// TwinCAT 3 PLC project Automation_BaseClasses
// Title: Automation base classes
// Company: PTW TUDa
// ProjectVersion: 0.1
// ProgramVersion: 3.1.4023.0
// project tree:
//   DUTs/0_Base Data Structs/ E_SystemControlState.TcDUT (not stored), E_SystemOperatingState.TcDUT (not stored), ST_Control.TcDUT (not stored), ST_ControlState.TcDUT (not stored), ST_ErrorState.TcDUT (not stored), ST_SetPointState.TcDUT, ST_SetSetPoint.TcDUT (not stored), ST_SystemState.TcDUT (not stored)
//   DUTs/Actor Data Structs/Pumps/ E_Liquids.TcTLEO, ST_PumpGrundfosMagna3SetParameters.TcDUT (not stored), ST_PumpGrundfosMagna3State.TcDUT (not stored)
//   DUTs/System Data Structs/ ST_SystemClimatizedRoomChillerSetParameters.TcDUT, ST_SystemClimatizedRoomChillerState.TcDUT
//   POUs/0_Base Clases/ FB_Actor2Point.TcPOU, FB_ActorContinous.TcPOU (not stored), FB_SystemContinous.TcPOU
//   POUs/Actors/ FB_PumpGrundfosMagna3.TcPOU
//   POUs/Sensors/ FB_AnalogSensor.TcPOU, FB_Flow_Sensor.TcPOU, FB_Pressure_Sensor.TcPOU, FB_Temp_Sensor.TcPOU (not stored)

// ---- DUTs/0_Base Data Structs/ST_SetPointState.TcDUT
{attribute 'OPC.UA.DA.StructuredType' := '1'}
TYPE ST_SetPointState :
STRUCT
	fOperatingPoint	: REAL; //current operating point
	fSetPoint		: REAL; //current set point
	aSetPointLimits	: ARRAY[1..2] OF REAL; //lower and upper limit of setpoint
END_STRUCT
END_TYPE

// ---- DUTs/Actor Data Structs/Pumps/E_Liquids.TcTLEO
{attribute 'qualified_only'}
{attribute 'strict'}
TYPE E_Liquids :
(
	water 	:= 0,
	glycol 	:= 1
);
END_TYPE

// ---- DUTs/System Data Structs/ST_SystemClimatizedRoomChillerSetParameters.TcDUT
{attribute 'OPC.UA.DA.StructuredType' := '1'}
TYPE ST_SystemClimatizedRoomChillerSetParameters :
STRUCT
	bDirectOperationOn 			: BOOL;
	bCondenserOn 				: BOOL;
END_STRUCT
END_TYPE

// ---- DUTs/System Data Structs/ST_SystemClimatizedRoomChillerState.TcDUT
{attribute 'OPC.UA.DA.StructuredType' := '1'}
TYPE ST_SystemClimatizedRoomChillerState :
STRUCT
	//general information
	bOperational				: BOOL;
	bErrorVentilator 			: BOOL;
	bErrorCompressor 			: BOOL;
	bErrorPump 					: BOOL;
	bErrorOverheatingControler 	: BOOL;
	
	//controler states
	bIR33ControlMode			: BOOL; // current control mode (0= proportional, 1= PID-control)
	nIR33OperatingMode			: INT; // current operating mode (1= Direct, 2= Reverse, 3= Neutralzone, 4= PWM, 5= Alarm, 6= Direct/Reverse over DI1, 7= Direct/Direct over DI1, 8= Reverse/Reverse over DI1, 9= Direct/Reverse with different set points)
	fIR33CurrentSetpointTemperature	: REAL; // Read setpoint temperature from controller
	bTemperatureUnit			: BOOL; // 0= °C, 1= °F
	
	//temperature sensors
	fTempSensorIR33		 		: REAL; //°C
	fTempCondenserAirIn 		: REAL; //°C
	fTempCondenserAirOut 		: REAL; //°C
	fTempCondenserMediumIn 		: REAL; //°C
	fTempCondenserMediumOut 	: REAL; //°C
	fTempCompressorSuctionLine 	: REAL; //°C
	fTempMediumIn 				: REAL; //°C
	fTempMediumOut 				: REAL; //°C
	
	//pressure sensors
	fPressureCondenserMediumOut 	: REAL; //bar
	fPressureCompressorSuctionLine 	: REAL; //bar
	
	//flow rate sensor
	fFlowRateMediumIn : REAL; //l/min
END_STRUCT
END_TYPE

// ---- POUs/0_Base Clases/FB_Actor2Point.TcPOU
FUNCTION_BLOCK ABSTRACT FB_Actor2Point
VAR_INPUT
	//internal input variables:
	bSetStatusOnAutomatic : BOOL; //turn actor on
	algorithmPermission : BOOL; //is true if control by algorithm is allowed
END_VAR
VAR_OUTPUT
END_VAR
VAR
	//OPC UA structured variables:
	{attribute 'OPC.UA.DA' := '1'}
	control : ST_Control;
	{attribute 'OPC.UA.DA' := '1'}
	controlState : ST_ControlState;
	{attribute 'OPC.UA.DA' := '1'}
	errorState : ST_ErrorState;
	
	//internal variables:
	bSetStatusOn : BOOL; //actual internal value to switch on 
END_VAR

METHOD PROTECTED SelectControlMode : BOOL
VAR_INPUT
END_VAR
//change access mode
IF control.bManualModeActivated THEN
	controlState.nAccessmode := E_SystemControlState.manual;
	controlState.sAccessMode := 'manual';
	bSetStatusOn := control.bSetStatusOnManual;
ELSIF control.bAlgorithmModeActivated AND algorithmPermission THEN
	controlState.nAccessmode := E_SystemControlState.algorithm;
	controlState.sAccessMode := 'algorithm';
	bSetStatusOn := control.bSetStatusOnAlgorithm;
ELSE
	controlState.nAccessmode := E_SystemControlState.automatic;
	controlState.sAccessMode := 'automatic';
	bSetStatusOn := bSetStatusOnAutomatic;
END_IF
END_METHOD

END_FUNCTION_BLOCK

// ---- POUs/0_Base Clases/FB_SystemContinous.TcPOU
FUNCTION_BLOCK ABSTRACT FB_SystemContinous EXTENDS FB_ActorContinous
VAR_INPUT
END_VAR
VAR_OUTPUT
END_VAR
VAR
	{attribute 'OPC.UA.DA' := '1'}
	systemState : ST_SystemState;
END_VAR

METHOD PROTECTED MAIN : BOOL // Method that calls all needed function block methods
VAR_INPUT
END_VAR
SUPER^.MAIN();
SystemFlowControl();
END_METHOD

METHOD PROTECTED ABSTRACT Operational : BOOL
VAR_INPUT
END_VAR
VAR_OUTPUT
	bSwitchToWorking : BOOL := FALSE;
END_VAR
END_METHOD

METHOD PROTECTED ABSTRACT RampDown : BOOL
VAR_INPUT
END_VAR
VAR_OUTPUT
	bRampDownFinished : BOOL := FALSE;
END_VAR
END_METHOD

METHOD PROTECTED ABSTRACT RampUp : BOOL
VAR_INPUT
END_VAR
VAR_OUTPUT
	bRampUpFinished : BOOL := FALSE;
END_VAR
END_METHOD

METHOD PROTECTED ABSTRACT StateCheck : BOOL
(* In this method the folowing elements of the actorState structrure have to be set if they are not set yet:
	bStatusOn 		: BOOL; //status on / off
	bError			: BOOL; //true if in error
	sErrorMessage	: STRING; //returns error message
	bWarning		: BOOL; //true if in warning
	sWarningMessage	: STRING; //returns warning message
	fOperatingPoint	: REAL; //current operating point
*)
VAR_INPUT
END_VAR
VAR
END_VAR
END_METHOD

METHOD SystemFlowControl : INT
VAR_INPUT
END_VAR
VAR_INST
	nState : E_SystemOperatingState := E_SystemOperatingState.standby; //actual state number
	bSwitchState : BOOL := FALSE;
END_VAR
CASE nState OF
	E_SystemOperatingState.standby:
		systemState.sOperatingState := 'standby';
		bSwitchState := FALSE;
		//if turned on switch to ramp-up
		IF(bSetStatusOn) THEN
			nState := E_SystemOperatingState.rampUp;
		END_IF
	E_SystemOperatingState.rampUp:
		systemState.sOperatingState := 'ramp-up';
		systemState.bRampUp := TRUE;
		RampUp(bRampUpFinished => bSwitchState);
		//if turned off switch to ramp-down
		IF(NOT bSetStatusOn) THEN
			nState := E_SystemOperatingState.rampDown;
		//if ramp-up finished switch to operational
		ELSIF(bSwitchState) THEN
			nState := E_SystemOperatingState.operational;
		END_IF
	E_SystemOperatingState.operational:
		systemState.sOperatingState := 'operational';
		Operational(bSwitchToWorking => bSwitchState);
		//if turned off switch to ramp-down
		IF(NOT bSetStatusOn) THEN
			nState := E_SystemOperatingState.rampDown;
		//switch to working if desired
		ELSIF(bSwitchState) THEN
			nState := E_SystemOperatingState.working;
		END_IF
	E_SystemOperatingState.working:
		systemState.sOperatingState := 'working';
		Working(bSwitchToOperational => bSwitchState);
		//if turned off switch to ramp-down
		IF(NOT bSetStatusOn) THEN
			nState := E_SystemOperatingState.rampDown;
		//switch to operational if desired
		ELSIF(bSwitchState) THEN
			nState := E_SystemOperatingState.operational;
		END_IF
	E_SystemOperatingState.rampDown:
		systemState.sOperatingState := 'ramp-down';
		systemState.bRampDown := TRUE;
		RampDown(bRampDownFinished => bSwitchState);
		//if turned on switch to ramp-up
		IF(bSetStatusOn) THEN
			nState := E_SystemOperatingState.rampUp;
		//if ramp-down finished switch to standby
		ELSIF(bSwitchState) THEN
			nState := E_SystemOperatingState.standby;
		END_IF
END_CASE
systemState.nOperatingState := nState;
END_METHOD

METHOD PROTECTED ABSTRACT Working : BOOL
VAR_INPUT
END_VAR
VAR_OUTPUT
	bSwitchToOperational : BOOL := FALSE;
END_VAR
END_METHOD

END_FUNCTION_BLOCK

// ---- POUs/Actors/FB_PumpGrundfosMagna3.TcPOU
FUNCTION_BLOCK FB_PumpGrundfosMagna3 EXTENDS FB_ActorContinous
VAR_INPUT
END_VAR
VAR_OUTPUT
END_VAR
VAR
	{attribute 'OPC.UA.DA' := '1'}
	localSetParameters : ST_PumpGrundfosMagna3SetParameters;
	{attribute 'OPC.UA.DA' := '1'}
	localState : ST_PumpGrundfosMagna3State;
	
	//external sensors connected
	bExternalTemperatureSensorConnected : BOOL := FALSE; //true if external temperature sensor connected
	bExternalFlowSensorConnected 		: BOOL := FALSE; //true if external flow sensor connected
	
	//I/O links
	fTemperatureInternalIn 		AT %I* : REAL; //°C
	fTemperatureExternalIn 		AT %I* : REAL; //°C external temperature from sensor connected to pump
	fTemperatureDifferenceIn	AT %I* : REAL; //°C
	fVolumeFlowRateIn 			AT %I* : REAL; //m^3/h volume flow rate from pump
	fPressureDifferenceIn	 	AT %I* : REAL; //pa = 10^-5 bar
	fPowerElectricIn			AT %I* : REAL; //W
	fPowerThermalIn	 			AT %I* : REAL; //W
	fRotationalSpeedIn	 		AT %I* : REAL; //rpm
END_VAR

MAIN();

//calculate thermal power if external sensors are connected
IF(bExternalTemperatureSensorConnected OR bExternalFlowSensorConnected) THEN
	CalculateThermalPower();
END_IF

METHOD PRIVATE CalculateThermalPower : BOOL
VAR_INPUT
END_VAR
VAR
	fMassFlowRate : REAL; //kg/s
	fDensity : REAL; // kg/m³
	fSpecificHeatCapacity : REAL; //J/(kg*K) 
	 
	fDensityWater : REAL := 997; // kg/m³
	fSpecificHeatCapacityWater : REAL := 4190; //J/(kg*K)
	fDensityGlycol : REAL := 1042; // kg/m³
	fSpecificHeatCapacityGlycol : REAL := 3400; //J/(kg*K)
END_VAR
CASE localState.nLiquid OF
	E_Liquids.water:
		fDensity := fDensityWater;
		fSpecificHeatCapacity := fSpecificHeatCapacityWater;
	E_Liquids.glycol:
		fDensity := fDensityGlycol;
		fSpecificHeatCapacity := fSpecificHeatCapacityGlycol;
END_CASE

fMassFlowRate := localState.fVolumeFlowRate / 60 * 0.001 * fDensity; //conversion from volume flow (l/min) to mass flow (kg/s)
localState.fPowerThermal :=  fMassFlowRate * localState.fTemperatureDifference * fSpecificHeatCapacity; //calculate thermal power
END_METHOD

METHOD ConnectExternalFlowSensor : BOOL
VAR_INPUT
	fExternalFlowValue : REAL; //l/min - input for external temperature value
END_VAR
VAR
END_VAR
bExternalFlowSensorConnected := TRUE;
localState.fVolumeFlowRate := fExternalFlowValue; //copy external sensor value to state
END_METHOD

METHOD ConnectExternalTemperatureSensor : BOOL
VAR_INPUT
	fExternalTemperatureValue : REAL; //input for external temperature value
END_VAR
bExternalTemperatureSensorConnected := TRUE;
localState.fTemperatureExternal := fExternalTemperatureValue; //copy external sensor value to state
localState.fTemperatureDifference := ABS(localState.fTemperatureInternal - localState.fTemperatureExternal); //calculate temperature difference
END_METHOD

END_FUNCTION_BLOCK

// ---- POUs/Sensors/FB_AnalogSensor.TcPOU
FUNCTION_BLOCK FB_AnalogSensor
VAR_INPUT
END_VAR
VAR_OUTPUT
	fValue 						: REAL; //converted sensor value
END_VAR
VAR
	nAnalogIn 			AT %I* 	: INT; //analog input value linked to real inputs
	fSensorlimitHigh 			: REAL; //upper limit of the sensor value range
	fSensorlimitLow 			: REAL; //lower limit of the sensor value range
	sUnit 						: STRING; //unit of the sensor value
END_VAR

fValue := ConvertedValue();

METHOD ConvertedValue : REAL
VAR_INPUT
END_VAR
// conversion from Bit value to actual value
ConvertedValue := ((INT_TO_REAL(nAnalogIn) / 32767 * (fSensorlimitHigh - fSensorlimitLow)) + fSensorlimitLow);
END_METHOD

METHOD FB_init : BOOL
VAR_INPUT
	bInitRetains : BOOL; // if TRUE, the retain variables are initialized (warm start / cold start)
	bInCopyCode : BOOL;  // if TRUE, the instance afterwards gets moved into the copy code (online change)
	fSensorlimitHigh : REAL; //upper limit of the sensor value range
	fSensorlimitLow : REAL; //lower limit of the sensor value range
	sUnit : STRING; //unit of the sensor value
END_VAR
//copy input values to internal variables
THIS^.fSensorlimitHigh := fSensorlimitHigh;
THIS^.fSensorlimitLow := fSensorlimitLow;
THIS^.sUnit := sUnit;
END_METHOD

END_FUNCTION_BLOCK

// ---- POUs/Sensors/FB_Flow_Sensor.TcPOU
FUNCTION_BLOCK FB_Flow_Sensor
VAR_INPUT
	flow_in AT %I* : INT;
END_VAR
VAR_OUTPUT
	flow_out : REAL;
END_VAR
VAR
	sensorlimit_high : REAL := 50.0;
	sensorlimit_low : REAL := 0.2;
END_VAR

// conversion from Bit value to temperature. 0 ~ 0,2 l/min, 32767 ~ 50 l/min
flow_out := (INT_TO_REAL(flow_in) / 32767 * (sensorlimit_high - sensorlimit_low)) + sensorlimit_low;

END_FUNCTION_BLOCK

// ---- POUs/Sensors/FB_Pressure_Sensor.TcPOU
FUNCTION_BLOCK FB_Pressure_Sensor
VAR_INPUT
	pressure_in AT %I* : INT;
END_VAR
VAR_OUTPUT
	pressure_out : REAL;
END_VAR
VAR
	sensorlimit_high : REAL := 90.0;
	sensorlimit_low : REAL := -30.0;
END_VAR

// conversion from Bit value to temperature. 0 ~ 2 bar, 32767 ~ 30 bar
pressure_out := (INT_TO_REAL(pressure_in) / 32767 * (sensorlimit_high - sensorlimit_low)) + sensorlimit_low;

END_FUNCTION_BLOCK
